_CFC_ (* Continuous Function Chart, elements in execution order *)
#0 <>(SHU6_PV1_M_MAXSPEED_CH, SHU6_PV1_M_MAXSPEED_CH_OLD)
#1 RS_RUCH:RS(SET: #0, RESET1: #3.Q)
#2 V_RUCH <= #1.Q1
#3 TON_RUCH:TON(IN: #1.Q1, PT: T#10s)
#4 SHU6_PV1_M_MAXSPEED <= SHU6_PV1_M_MAXSPEED_CH
#5 AND(SHU6_PV1_YA3_M_UST_VKL_UVEL_CHAST, SHU6_PV1_YA4_M_UST_VKL_UVEL_CHAST, SHU6_PV1_UST_RE_RABOTA)
#6 TON_STER_1:TON(IN: #5, PT: T#60s)
#7 OR(#6.Q, SHU6_PV1_M_SB2_STER_REG)
#8 AND(#7, SHU6_PV1_UST_RE_RABOTA, NOT V_RUCH)
#9 OR(V_RUCH, SHU6_PV1_UST_RE_PUSK)
#10 SEL(#8, SHU6_PV1_SPEEDMOTOR, SHU6_PV1_M_MAXSPEED)
#11 AND(#8, NOT V_RUCH)
#12 SEL(#11, SHU6_PV1_M_USKORENIE_PUSK, SHU6_PV1_M_USKORENIE_UPR)
#13 OR(SHU6_PV1_YA3_B_UST_VKL_STER_REG, SHU6_PV1_YA4_B_UST_VKL_STER_REG)
#14 AND(SHU6_PV1_UST_RE_RABOTA, #13)
#15 TON_STER_2:TON(IN: #14, PT: T#60s)
#16 AND(NOT SHU6_PV1_M_SB2_STER_REG, #15.Q, SHU6_PV1_UST_RE_RABOTA, NOT V_RUCH)
#17 SEL(#16, #10, SHU6_PV1_M_MINSPEED)
#18 SEL(#9, #17, SHU6_PV1_M_MAXSPEED)
#19 SEL(SHU6_PV1_UST_SOST_VKL, 0, #18)
#20 AND(#16, NOT V_RUCH)
#21 SEL(#20, SHU6_PV1_M_ZAMEDLENIE_OST, SHU6_PV1_M_ZAMEDLENIE_UPR)
#22 SEL(SHU6_PV1_UST_SET_STOP, #21, 1000)
#23 RR:RAMP_REAL(#19, #12, #22, T#1s, -)
#24 SHU6_PV1_SPEEDMOTOR <= #23
#25 SHU6_PV1_M_MAXSPEED_CH_OLD <= SHU6_PV1_M_MAXSPEED_CH
#26 RT_KOMVKL_2:R_TRIG(CLK: TRUE)
#27 MOVE(EN: #26.Q, 5)
#28 SHU6_PV1_MP1_ZAD_RUCH <= #27
#29 RT_KOMVKL_3:R_TRIG(CLK: TRUE)
#30 MOVE(EN: #29.Q, 5)
#31 SHU6_PV1_MV1_ZAD_RUCH <= #30
#32 MOVE(EN: SHU6_PV1_MP1_DO1_VKL, #23)
#33 SEL(#32.ENO, 0, #32)
#34 SEL(SHU6_PV1_SA1MP1_DI6_M, #33, SHU6_PV1_MP1_ZAD_RUCH)
#35 SHU6_PV1_MP1_ZAD_VN <= #34
#36 MOVE(EN: SHU6_PV1_MV1_DO3_VKL, #23)
#37 SEL(#36.ENO, 0, #36)
#38 SEL(SHU6_PV1_YAMV1_DI8_M, #37, SHU6_PV1_MV1_ZAD_RUCH)
#39 SHU6_PV1_MV1_ZAD_VN <= #38
_END_CFC_
END_PROGRAM

(* POU IM/MRQ1_Upr, CFC *)
PROGRAM MRQ1_Upr
VAR

	tTi: TIME;
	tTv: TIME := T#0s;
	tTd: TIME := T#0s;

	startDelay_M3: TIME := T#0s;
	stopDelay_M3: TIME := T#0s;
	delayFBC_M3: TIME := T#30S;
	feedbPT_M3: TIME := T#120s;
	delayFBP_M3: TIME := T#30s;

	fb_HVACMS_M3: FB_HVACMotor1Speed;
	SR_VKL: SR;
END_VAR
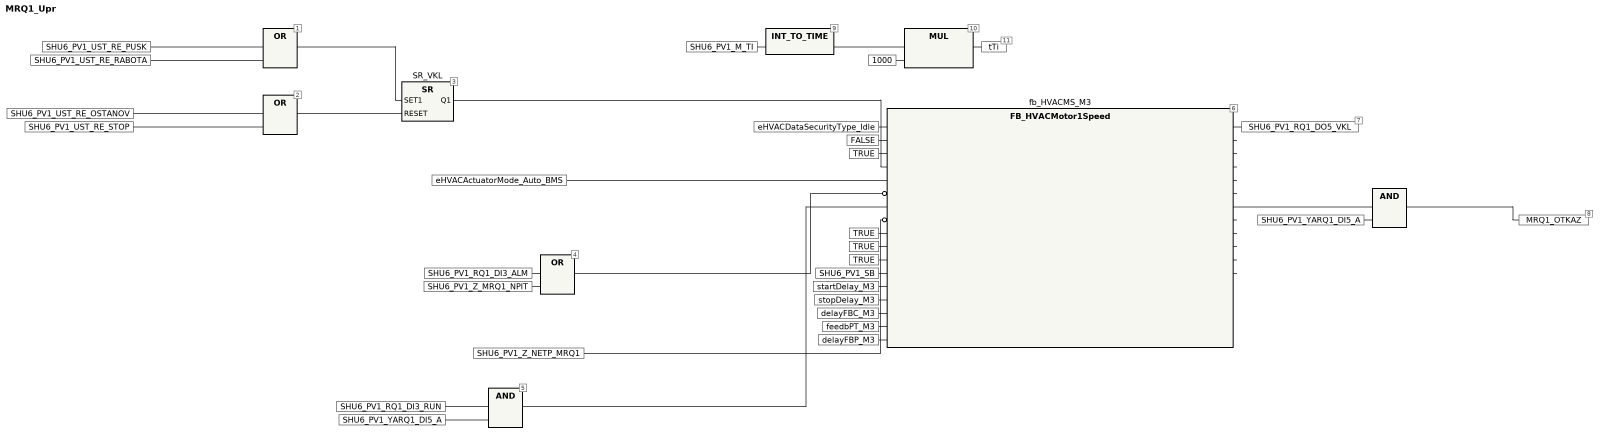
